Fanuc KAREL source: ko00054.KL

-- PROVISIONAL review KL for V1013-1; original PC SHA256 b603e9ae3018ece86fd8e3cfb8b0d975c94ce529756be6f5937eecf88e03e23b
-- Incomplete behavior may be omitted. Consult companion uncertainty JSON. Do not deploy.
PROGRAM KO00054
%NOLOCKGROUP
BEGIN
  -- UNRESOLVED_PC offsets 5-12; opcodes 9D,23
  -- UNRESOLVED_PC offsets 17-69; opcodes 27,27,49,7E,AD,27,49,7E,AD,22,31,7E,4A
  -- UNRESOLVED_PC offsets 74-78; opcodes 7F
END KO00054
